FUNCTION_BLOCK FB_Testcase IMPLEMENTS I_Testcase
VAR_INPUT
	nNumber:			INT:= E_Number.Init;
	sName:				STRING(255);	//	name        The name of this test case, often the method name  
	sClassname:			STRING(255);	//	classname   The name of the parent class/folder, often the same as the suite's name
	nAssertions:		INT; 			//	assertions  Number of assertions checked during test case execution  
	fTime:				LREAL;			//	time        Execution time of the test in seconds            
	sFile:				STRING(255);	//	file        Source code file of this test case              
	nLine:				INT;			//	line        Source code line number of the start of this test case  	
END_VAR
VAR_OUTPUT
END_VAR
VAR
END_VAR

METHOD PUBLIC M_Switch
VAR_INPUT
	Next:				INT;			// Next test case
END_VAR
sName:= '';
sClassname:= '';
nAssertions:= 0;
fTime:= 0.0;
sFile:= '';
nLine:= 0;
nNumber:= Next;
END_METHOD

PROPERTY PUBLIC P_Assertions : INT
GET
P_Assertions:= nAssertions;
END_GET
SET
nAssertions:= P_Assertions;
END_SET
END_PROPERTY

PROPERTY PUBLIC P_Classname : STRING(255)
GET
P_Classname:= sClassname;
END_GET
SET
sClassname:= P_Classname;
END_SET
END_PROPERTY

PROPERTY PUBLIC P_File : STRING(255)
GET
P_File:= sFile;
END_GET
SET
sFile:= P_File;
END_SET
END_PROPERTY

PROPERTY PUBLIC P_Line : INT
GET
P_Line:= nLine;
END_GET
SET
nLine:= P_Line;
END_SET
END_PROPERTY

PROPERTY PUBLIC P_Name : STRING(255)
GET
P_Name:= sName;
END_GET
SET
sName:= P_Name;
END_SET
END_PROPERTY

PROPERTY PUBLIC P_Number : Int
GET
P_Number:= nNumber;
END_GET
SET
nNumber:= P_Number;
END_SET
END_PROPERTY

PROPERTY PUBLIC P_Time : Lreal
GET
P_Time:= fTime;
END_GET
SET
fTime:= P_Time;
END_SET
END_PROPERTY

END_FUNCTION_BLOCK

(* stored: Version 1.1.0.1
   POU FB_Testcase: Id {8a94cda9-7d7f-4f18-843a-69c57a60ec24}, SpecialFunc None
   Method M_Switch: Id {1c98ed0f-b19e-47ad-9b6d-976810c9e896}
   Property P_Assertions: Id {686f81f2-34eb-4b3b-81a3-02e245ca80f9}
   Get Get: Id {9617c176-29fa-45a0-b937-39e6e799cde0}
   Set Set: Id {ad1111a1-fe21-4e8b-9000-85ad29de187a}
   Property P_Classname: Id {390cee0a-010d-4204-b1b1-9129bc6413c1}
   Get Get: Id {2688e1f2-e3e8-4245-80d2-74b152c9ca9c}
   Set Set: Id {55b3dd43-1cda-4eae-b750-9bc915384faa}
   Property P_File: Id {b2c2210b-f780-4e46-81e5-f39e00341986}
   Get Get: Id {8edcc67f-7ccd-4392-84e3-e6479a44e142}
   Set Set: Id {5763219c-f732-4b54-8014-5903946a2a6a}
   Property P_Line: Id {cc49a74c-be9b-4859-a563-dba1e6ecf2da}
   Get Get: Id {c3e11b66-8047-4b92-9339-469885dbdc1b}
   Set Set: Id {42183ec2-002d-43e0-9f41-3cf0c99bb621}
   Property P_Name: Id {f64f135e-18bc-4bda-a3f6-2563788f034f}
   Get Get: Id {c2f5088a-1ba2-4d42-83a7-dbed764bd892}
   Set Set: Id {d7365e50-2600-4659-b7f7-8e28548f6d09}
   Property P_Number: Id {a5d185c8-a21f-418f-b65c-f3bb459e57ca}
   Get Get: Id {3a4e05cd-0a11-46d0-8882-d1094443319f}
   Set Set: Id {c54591f4-5e3a-43eb-a3ff-0ba3a1e50fa1}
   Property P_Time: Id {2fdcf9da-b796-4097-9b53-b145e25f0025}
   Get Get: Id {0ce03ffb-e6ea-4959-b011-cc36e6dcb2d1}
   Set Set: Id {9d548146-a437-4646-96bb-98cf58cefe79} *)
